FUNCTION_BLOCK SEND_LINE_DATA (* Send linear movement data *)
  (* Standard: 61499-2 *)
  (* Version 1.0, 17-04-2012, GASR, Universidade do Estado de Santa Catarina *)
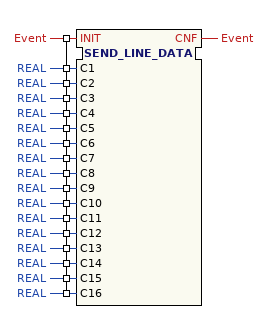
  EVENT_INPUT
    INIT WITH C1, C2, C3, C4, C5, C6, C7, C8, C9, C10, C11, C12, C13, C14, C15, C16;
  END_EVENT
  EVENT_OUTPUT
    CNF;
  END_EVENT
  VAR_INPUT
    C1 : REAL; (* Coeficient 1 *)
    C2 : REAL; (* Coeficient 2 *)
    C3 : REAL; (* Coeficient 3 *)
    C4 : REAL; (* Coeficient 4 *)
    C5 : REAL; (* Coeficient 5 *)
    C6 : REAL; (* Coeficient 6 *)
    C7 : REAL; (* Coeficient 7 *)
    C8 : REAL; (* Coeficient 8 *)
    C9 : REAL; (* Coeficient 9 *)
    C10 : REAL; (* Coeficient 10 *)
    C11 : REAL; (* Coeficient 11 *)
    C12 : REAL; (* Coeficient 12 *)
    C13 : REAL; (* Coeficient 13 *)
    C14 : REAL; (* Coeficient 14 *)
    C15 : REAL; (* Coeficient 15 *)
    C16 : REAL; (* Coeficient 16 *)
  END_VAR
  FBS
    set_line_data : SET_LINE_DATA;
    comm_all_axel : GENERAL_DATA_SENDER;
    comm_x : AXIS_DATA_SENDER;
    comm_y : AXIS_DATA_SENDER;
    comm_z : AXIS_DATA_SENDER;
  END_FBS
  EVENT_CONNECTIONS
    INIT TO set_line_data.INIT;
    set_line_data.CNF TO comm_all_axel.INIT;
    comm_x.CNF TO comm_y.INIT;
    comm_y.CNF TO comm_z.INIT;
    comm_z.CNF TO CNF;
    comm_all_axel.CNF TO comm_x.INIT;
  END_CONNECTIONS
  DATA_CONNECTIONS
    C16 TO set_line_data.C16;
    C13 TO set_line_data.C13;
    C15 TO set_line_data.C15;
    C11 TO set_line_data.C11;
    C6 TO set_line_data.C6;
    C7 TO set_line_data.C7;
    C4 TO set_line_data.C4;
    C5 TO set_line_data.C5;
    C12 TO set_line_data.C12;
    C14 TO set_line_data.C14;
    C9 TO set_line_data.C9;
    C8 TO set_line_data.C8;
    C1 TO set_line_data.C1;
    C10 TO set_line_data.C10;
    C3 TO set_line_data.C3;
    C2 TO set_line_data.C2;
    set_line_data.ax_1 TO comm_x.SD_1;
    set_line_data.ax_2 TO comm_x.SD_2;
    set_line_data.Vx_2 TO comm_x.SD_6;
    set_line_data.bx_1 TO comm_x.SD_3;
    set_line_data.Vx_1 TO comm_x.SD_5;
    set_line_data.id TO comm_x.ID;
    set_line_data.bx_2 TO comm_x.SD_4;
    set_line_data.ay_1 TO comm_y.SD_1;
    set_line_data.ay_2 TO comm_y.SD_2;
    set_line_data.Vy_2 TO comm_y.SD_6;
    set_line_data.by_1 TO comm_y.SD_3;
    set_line_data.Vy_1 TO comm_y.SD_5;
    set_line_data.id TO comm_y.ID;
    set_line_data.by_2 TO comm_y.SD_4;
    set_line_data.az_1 TO comm_z.SD_1;
    set_line_data.az_2 TO comm_z.SD_2;
    set_line_data.Vz_2 TO comm_z.SD_6;
    set_line_data.bz_1 TO comm_z.SD_3;
    set_line_data.Vz_1 TO comm_z.SD_5;
    set_line_data.id TO comm_z.ID;
    set_line_data.bz_2 TO comm_z.SD_4;
    set_line_data.t0 TO comm_all_axel.SD_1;
    set_line_data.t TO comm_all_axel.SD_2;
    set_line_data.speed_1 TO comm_all_axel.SD_3;
    set_line_data.id TO comm_all_axel.ID;
    set_line_data.speed_2 TO comm_all_axel.SD_4;
  END_CONNECTIONS
END_FUNCTION_BLOCK
